// TwinCAT 3 PLC project plc_vat_test
// ProgramVersion: 3.1.4024.12
// libraries:
//   LCLS General, * (SLAC)
//   PMPS, * (SLAC - LCLS)
//   Tc2_EtherCAT, * (Beckhoff Automation GmbH)
//   Tc2_Math, * (Beckhoff Automation GmbH)
//   Tc2_Standard, * (Beckhoff Automation GmbH)
//   Tc2_System, * (Beckhoff Automation GmbH)
//   Tc2_Utilities, * (Beckhoff Automation GmbH)
//   Tc3_Module, * (Beckhoff Automation GmbH)
//   LCLS Vacuum,newest,SLAC - LCLS
// project tree:
//   DUTs/ ST_CoeParamsTest.TcDUT
//   DUTs/VAT590/EtherCAT Interface/ E_ControlMode.TcDUT, E_ControlModeSP.TcDUT (not stored), E_FatalErrors.TcDUT, ST_ExtendedWarnings.TcDUT (not stored), ST_GeneralControlSP.TcDUT (not stored), ST_GeneralStatus.TcDUT (not stored), ST_GeneralWarnings.TcDUT (not stored)
//   DUTs/VAT590/ E_VAT590_PID_CTRL.TcDUT (not stored), E_VAT590_PressureSensor.TcDUT (not stored), E_VCN_VAT590.TcDUT (not stored), E_VAT590_AccessMode.TcDUT (not stored), ST_CoEIndSub.TcDUT (not stored), ST_VAT590_COE.TcDUT, ST_VCN_VAT590.TcDUT, ST_VAT590_STATUS.TcDUT (not stored)
//   GVLs/ GVL_IO.TcGVL
//   / PlcTask.TcTTO
//   POUs/CoE/ FB_CoE_Read.TcPOU, FB_CoE_Write.TcPOU
//   POUs/Gauges/ FB_IE514.TcPOU, FB_MX7M.TcPOU
//   POUs/Valves/ FB_VCN_VAT590.TcPOU
//   POUs/ MAIN.TcPOU
// real-time tasks:
//   TASK PlcTask: cycle T#10ms, priority 20, ADS port 350
// I/O:
//   DEVICE Device 1 (EtherCAT), AmsNetId 172.21.132.149.2.1
//     Term 1 (EK1200) [EK1200-5000 EtherCAT Power supply (2A E-Bus)]
//       Term 3 (EL1004) [EL1004 4Ch. Dig. Input 24V, 3ms]
//       Term 5 (EL3174-0002) [EL3174-0002 4Ch. Ana. Input +/-10V, +/-20mA 16 Bit, Isolated Channels]
//       Term 10 (EL2624) [EL2624 4Ch. Relay Output, NO (125V AC / 30V DC)]
//       Term 8 (EK1110) [EK1110 EtherCAT extension]
//     VAT590_TEST [590 - All-metal variable leak valve]
// variable links:
//   plc_vat_test/plc_vat_test Instance <-> Device 1 (EtherCAT)/Term 1 (EK1200)/Term 10 (EL2624)
//     PlcTask Outputs/MAIN.fbIE514.q_xHV_DIS_CH1 <-> Channel 1/Output
//     PlcTask Outputs/MAIN.fbIE514.q_xHV_DIS_CH2 <-> Channel 2/Output
//     PlcTask Outputs/MAIN.fbMX7M.q_xHV_DIS <-> Channel 3/Output
//   plc_vat_test/plc_vat_test Instance <-> Device 1 (EtherCAT)/Term 1 (EK1200)/Term 3 (EL1004)
//     PlcTask Inputs/MAIN.fbIE514.i_xCH2_SEL <-> Channel 2/Input
//     PlcTask Inputs/MAIN.fbIE514.i_xERR_CH1 <-> Channel 3/Input
//     PlcTask Inputs/MAIN.fbIE514.i_xERR_CH2 <-> Channel 4/Input
//     PlcTask Inputs/MAIN.fbIE514.i_xHV_ON <-> Channel 1/Input
//   plc_vat_test/plc_vat_test Instance <-> Device 1 (EtherCAT)/Term 1 (EK1200)/Term 5 (EL3174-0002)
//     PlcTask Inputs/MAIN.fbIE514.i_iPRESS_R <-> AI Standard Channel 1/Value
//     PlcTask Inputs/MAIN.fbMX7M.i_iPRESS_R <-> AI Standard Channel 3/Value
//   plc_vat_test/plc_vat_test Instance <-> Device 1 (EtherCAT)/VAT590_TEST
//     PlcTask Inputs/MAIN.fbVCN590.i_bValveEthCatStatus <-> WcState/WcState
//     PlcTask Inputs/MAIN.fbVCN590.i_eControlMode <-> DI TxPDO-Map/Control mode
//     PlcTask Inputs/MAIN.fbVCN590.i_eFatalError <-> DI TxPDO-Map/Fatal error
//     PlcTask Inputs/MAIN.fbVCN590.i_nRawPosition <-> DI TxPDO-Map/Position
//     PlcTask Inputs/MAIN.fbVCN590.i_nRawPressure <-> DI TxPDO-Map/Pressure
//     PlcTask Inputs/MAIN.fbVCN590.i_stExtnWarnings <-> DI TxPDO-Map/Extended warnings
//     PlcTask Inputs/MAIN.fbVCN590.i_stGenStatus <-> DI TxPDO-Map/General status
//     PlcTask Inputs/MAIN.fbVCN590.i_stGenWarnings <-> DI TxPDO-Map/General warnings
//     PlcTask Inputs/MAIN.fbVCN590.i_stVat590PlcDriveRef/aNetId <-> InfoData/AdsAddr/netId
//     PlcTask Inputs/MAIN.fbVCN590.i_stVat590PlcDriveRef/nSlaveAddr <-> InfoData/AdsAddr/port
//     PlcTask Outputs/MAIN.fbVCN590.o_eCtrlModeSP <-> DO RxPDO-Map/Control mode setpoint
//     PlcTask Outputs/MAIN.fbVCN590.o_nRawPositionSP <-> DO RxPDO-Map/Position setpoint
//     PlcTask Outputs/MAIN.fbVCN590.o_nRawPressureSP <-> DO RxPDO-Map/Pressure setpoint
//     PlcTask Outputs/MAIN.fbVCN590.o_stGenCtrlSP <-> DO RxPDO-Map/General control setpoint

CONFIGURATION plc_vat_test
    RESOURCE PLC ON TwinCAT3
        TASK PlcTask(INTERVAL := T#10ms, PRIORITY := 20);
        PROGRAM MAIN WITH PlcTask : MAIN;
    END_RESOURCE
END_CONFIGURATION

// ---- DUTs/ST_CoeParamsTest.TcDUT
TYPE ST_CoeParamsTest :
STRUCT
	nWarnTemp : BYTE;
	nSwOffTemp : BYTE;
	nOffestA : INT;
	nOffestB : INT;
END_STRUCT
END_TYPE

// ---- DUTs/VAT590/EtherCAT Interface/E_ControlMode.TcDUT
{attribute 'qualified_only'}
{attribute 'strict'}
TYPE E_ControlMode :
(
	Init := 0,
	Synch := 1,
	ManualControl := 2,
	CloseValve := 3,
	OpenValve := 4,
	PressureControl := 5,
	HoldValve := 6,
	LearnProcedure := 7,
	InterlockOpen := 8,
	InterlockClose := 9,
	MaintenanceOpen := 10,
	MaintenanceClose := 11,
	PowerFailure := 12,
	Safety := 13,
	FatalError := 14
) USINT;
END_TYPE

// ---- DUTs/VAT590/EtherCAT Interface/E_FatalErrors.TcDUT
{attribute 'qualified_only'}
{attribute 'strict'}
TYPE E_FatalErrors :
(
	NO_FATAL_ERROR := 0,
	NoStopDetectedSynch := 20,
	ValveBlockedSynch := 21,
	ValveBlocked := 22,
	StepLossSynch := 25,
	MotorDriverFault := 40
) UINT;
END_TYPE

// ---- DUTs/VAT590/ST_VAT590_COE.TcDUT
TYPE ST_VAT590_COE :
STRUCT
	{attribute 'pytmc' := '
	pv: PID_CTRL
	io: io
	'}
	ePIDCtrl: E_VAT590_PID_CTRL;
	(*Adaptive Downstream Parameters*)
	{attribute 'pytmc' := '
    pv: SENS_DELAY_AD
	io: io
	field: EGU "s"
	field: DRVL 0.0
	field: DRVH 1.0
    '}
	fSensorDelay_AD : REAL;
	{attribute 'pytmc' := '
    pv: RAMP_TIME_AD
	io: io
	field: EGU "s"
	field: DRVL 0.0
	field: DRVH 1000000.0
    '}
	fRampTime_AD : REAL;
	{attribute 'pytmc' := '
    pv: RAMP_MODE_AD
	io: io
	field: ZNAM CONST_TIME
	field: ONAM CONST_SLOPE
    '}
	nRampMode_AD : BOOL;
	{attribute 'pytmc' := '
    pv: GAIN_FACTOR_AD
	io: io
	field: PREC 4
	field: DRVL 0.0001
	field: DRVH 7.5
    '}
	fGainFactor_AD : REAL;
	(*Fixed 1 Parameters*)
	{attribute 'pytmc' := '
    pv: RAMP_TIME_FIX1
	io: io
	field: EGU "s"
	field: DRVL 0.0
	field: DRVH 1000000.0
    '}
	fRampTime_FIX1 : REAL;
	{attribute 'pytmc' := '
    pv: RAMP_MODE_FIX1
	io: io
	field: ZNAM CONST_TIME
	field: ONAM CONST_SLOPE
    '}
	nRampMode_FIX1 : BOOL;
	{attribute 'pytmc' := '
    pv: CTRL_DIR_FIX1
	io: io
	field: ZNAM DOWNSTREAM
	field: ONAM UPSTREAM
    '}
	nCtrlDir_FIX1 : BOOL;
	{attribute 'pytmc' := '
    pv: PGAIN_FIX1
	io: io
	field: DRVL 0.001
	field: DRVH 100.0
    '}
	fPGain_FIX1 : REAL;
	{attribute 'pytmc' := '
    pv: IGAIN_FIX1
	io: io
	field: DRVL 0.0
	field: DRVH 100.0
    '}
	fIGain_FIX1 : REAL;
	(*Fixed 2 Parameters*)
	{attribute 'pytmc' := '
    pv: RAMP_TIME_FIX2
	io: io
	field: EGU "s"
	field: DRVL 0.0
	field: DRVH 1000000.0
    '}
	fRampTime_FIX2 : REAL;
	{attribute 'pytmc' := '
    pv: RAMP_MODE_FIX2
	io: io
	field: ZNAM CONST_TIME
	field: ONAM CONST_SLOPE
    '}
	nRampMode_FIX2 : BOOL;
	{attribute 'pytmc' := '
    pv: CTRL_DIR_FIX2
	io: io
	field: ZNAM DOWNSTREAM
	field: ONAM UPSTREAM
    '}
	nCtrlDir_FIX2 : BOOL;
	{attribute 'pytmc' := '
    pv: PGAIN_FIX2
	io: io
	field: DRVL 0.001
	field: DRVH 100.0
    '}
	fPGain_FIX2 : REAL;
	{attribute 'pytmc' := '
    pv: IGAIN_FIX2
	io: io
	field: DRVL 0.0
	field: DRVH 100.0
    '}
	fIGain_FIX2 : REAL;
	(*Soft Pump Parameters*)
	{attribute 'pytmc' := '
    pv: RAMP_TIME_SP
	io: io
	field: EGU "s"
	field: DRVL 0.0
	field: DRVH 1000000.0
    '}
	fRampTime_SP : REAL;
	{attribute 'pytmc' := '
    pv: RAMP_MODE_SP
	io: io
	field: ZNAM CONST_TIME
	field: ONAM CONST_SLOPE
    '}
	nRampMode_SP : BOOL;
	{attribute 'pytmc' := '
    pv: PGAIN_SP
	io: io
	field: DRVL 0.001
	field: DRVH 100.0
    '}
	fPGain_SP : REAL;
END_STRUCT
END_TYPE

// ---- DUTs/VAT590/ST_VCN_VAT590.TcDUT
TYPE ST_VCN_VAT590 :
STRUCT
	(* VCN - Valve Controlled Needle
	Used for VAT590 needle valves *)
	{attribute 'pytmc' := '
    pv: POS_RAW
	io: i
    '}
	nRawPosition : DINT; //Position readback
	{attribute 'pytmc' := '
    pv: PRES_RAW
	io: i
    '}
	nRawPressure : DINT; //Pressure readback
	{attribute 'pytmc' := '
    pv: PRES_TORR
	field: EGU "TORR"
	io: i
    '}
	fPressure : REAL; //Pressure readback in Torr units
	{attribute 'pytmc' := '
	pv: POS_SP
	io: i
	'}
	nPositionSP : DINT; //Position setpoint readback
	{attribute 'pytmc' := '
	pv: PRES_SP
	io: i
	'}
	nPressureSP : DINT; //Pressure setpoint readback
	{attribute 'pytmc' := '
    pv: ILK_OK
	field: ZNAM NOT OK
	field: ONAM OK
	field: ZSV MAJOR
	field: OSV NO_ALARM
	io: i
    '}
	bIlkOK : BOOL := FALSE; // Interlock Bit status
	{attribute 'pytmc' := '
    pv: POS_LIMIT
	io: io
	autosave_pass1: VAL DESC
    '}
	fPosSetLimit	: REAL := 100; // Percentage Upper limit on valve open
	{attribute 'pytmc' := '
    pv: PRES_SET_LIMIT
	io: io
	autosave_pass1: VAL DESC
    '}
	fPresSetLimit	: REAL := 1E-2; // Upper limit for pressure control 	
	{attribute 'pytmc' := '
    pv: PRES_RDBK_LIMIT
	io: io
	autosave_pass1: VAL DESC
    '}	
	fPresRdbkLimit : REAL := 1E-4;  //upper limit for pressure reading before valve close
	{attribute 'pytmc' := '
	pv: POS_REQ
	field: DRVL 0.0
	field: DRVH 100.0
	io: io
	'}
	fReqPosition : REAL; //Requested position (0.0-100.0%)
	{attribute 'pytmc' := '
	pv: PRES_REQ
	field: EGU "TORR"
	io: io;
	'}
	fReqPressure : REAL; //Requested pressure in Torr units
	{attribute 'pytmc' :=  ' 
	pv: STATE
	io: io
	'}
	eValveControl : E_VCN_VAT590; //Valve control mode
	{attribute 'pytmc' := '
    pv: 
	'}
	stValveStatus : ST_VAT590_STATUS; //All Valve status readbacks
	{attribute 'pytmc' :=  ' 
	pv: PRES_SENS
	io: io
	'}
	ePressureSensor : E_VAT590_PressureSensor; // Select pressure sensor
	{attribute 'pytmc' :=  ' 
	pv: REM_CTRL
	io: o
	'}
	eRemoteControl : E_VAT590_AccessMode; // Select remote control mode
	{attribute 'pytmc' := '
	pv: ZERO
	field: ZNAM NOT_ACTIVE
	field: ONAM ACTIVE
	io: o
	'}
	bZero : BOOL; // Activate Zero function bit
	{attribute 'pytmc' := '
    pv: 
	'}
	stCoeParameters : ST_VAT590_COE; //Coe Parameters
	{attribute 'pytmc' := '
	pv: COE_ERROR
	io: i
	field: ZNAM OK
	field: ONAM ERROR
	field: ZSV NO_ALARM
	field: OSV MAJOR
	'}
	bCoeError : BOOL; //Coe Interface Error
	{attribute 'pytmc' := '
	pv: COE_RESET
	io: io
	'}
	bResetCoeError : BOOL; //Reset Coe Interface
END_STRUCT
END_TYPE

// ---- GVLs/GVL_IO.TcGVL
{attribute 'qualified_only'}
VAR_GLOBAL
	//stPlcDriveRef AT %I*: ST_PlcDriveRef;
END_VAR

// ---- POUs/MAIN.TcPOU
PROGRAM MAIN
VAR
	
    {attribute 'pytmc' := '
      pv: VCN:TEST:01
    '}
	fbVCN590 : FB_VCN_VAT590; // Variable leak valve VAT590 function block
	fbMKS500 : FB_MKS500;
	
	stVG : ST_VG;
    {attribute 'pytmc' := '
      pv: GHC:TEST
    '}
	fbIE514 : FB_IE514;
	
    {attribute 'pytmc' := '
      pv: GCC:TEST
    '}
	fbMX7M : FB_MX7M;
	rPiraniPressure : REAL := 1E-4;
	
	rRealNumber : REAL := 8.367;
	intPart: INT;
    fracPart: REAL;
	rPressure : REAL := 0;
END_VAR

stVG.xPRESS_OK := TRUE;
stVG.rPress := rPiraniPressure;
fbMKS500.M_SetBits(30518);
fbMKS500(PG := stVG);

fbVCN590(bExtIlkOK := TRUE, IG := stVG);

fbIE514(PG := stVG);

fbMX7M(PG := stVG);

intPart := TRUNC_INT(rRealNumber); // Get the integer part
fracPart := LREAL_TO_REAL(FRAC(rRealNumber)); // Get the fractional part

rPressure := fracPart * LREAL_TO_REAL(EXPT(10,(intPart-11)));

END_PROGRAM

// ---- POUs/Valves/FB_VCN_VAT590.TcPOU
(* This function implements the Basic functions for the VAT590 needle valve*)
FUNCTION_BLOCK FB_VCN_VAT590 EXTENDS FB_Valve
VAR_INPUT
	bExtIlkOK : BOOL;        // External Interlock, SET to TRUE if not used
	IG : ST_VG;              // Input from a cold cathode gauge used in control loop
END_VAR
VAR_OUTPUT
	{attribute 'pytmc' := '
    pv:
	'}
	stVcnVat590	: ST_VCN_VAT590;       // Needle valve VAT590 structure
END_VAR
VAR CONSTANT
	cOpenPosition : REAL := 1E+5;      // Default position setpoint upper scale value
	cClosePosition : REAL := 0.0;      // Default position setpoint lower scale value
	cPresSPUpLim : REAL := 1E+6;       // Default pressure setpoint upper scale value
	cPresSPLowLim : REAL := 0;         // Default pressure setpoint lower scale value
	cPressCtrl : ST_CoEIndSub := (nIndex := 16#2199, nSubIndex := 0); // Selected pressure controller CoE register
	cSensorDelay_AD : ST_CoEIndSub := (nIndex := 16#219A, nSubIndex := 0); // Adaptive DS controller Sensor Delay CoE register
	cRampTime_AD : ST_CoEIndSub := (nIndex := 16#219B, nSubIndex := 0); // Adaptive DS controller Ramp Time CoE register
	cRampMode_AD : ST_CoEIndSub := (nIndex := 16#219C, nSubIndex := 0); // Adaptive DS controller Ramp Mode CoE register
	cGainFactor_AD : ST_CoEIndSub := (nIndex := 16#219E, nSubIndex := 0); // Adaptive DS controller Gain factor CoE register
	cRampTime_FIX1 : ST_CoEIndSub := (nIndex := 16#21A5, nSubIndex := 0); // Fixed 1 controller Ramp Time CoE register
	cRampMode_FIX1 : ST_CoEIndSub := (nIndex := 16#21A6, nSubIndex := 0); // Fixed 1 controller Ramp Mode CoE register
	cCtrlDir_FIX1 : ST_CoEIndSub := (nIndex := 16#21A7, nSubIndex := 0); // Fixed 1 controller Control Direction CoE register
	cPGain_FIX1 : ST_CoEIndSub := (nIndex := 16#21A8, nSubIndex := 0); // Fixed 1 controller P Gain CoE register
	cIGain_FIX1 : ST_CoEIndSub := (nIndex := 16#21A9, nSubIndex := 0); // Fixed 1 controller I Gain CoE register
	cRampTime_FIX2 : ST_CoEIndSub := (nIndex := 16#21AF, nSubIndex := 0); // Fixed 2 controller Ramp Time CoE register
	cRampMode_FIX2 : ST_CoEIndSub := (nIndex := 16#21B0, nSubIndex := 0); // Fixed 2 controller Ramp Mode CoE register
	cCtrlDir_FIX2 : ST_CoEIndSub := (nIndex := 16#21B1, nSubIndex := 0); // Fixed 2 controller Control Direction CoE register
	cPGain_FIX2 : ST_CoEIndSub := (nIndex := 16#21B2, nSubIndex := 0); // Fixed 2 controller P Gain CoE register
	cIGain_FIX2 : ST_CoEIndSub := (nIndex := 16#21B3, nSubIndex := 0); // Fixed 2 controller I Gain CoE register
	cRampTime_SP : ST_CoEIndSub := (nIndex := 16#21B9, nSubIndex := 0); // Soft Pump controller Ramp Time CoE register
	cRampMode_SP : ST_CoEIndSub := (nIndex := 16#21BA, nSubIndex := 0); // Soft Pump controller Ramp Time CoE register
	cPGain_SP : ST_CoEIndSub := (nIndex := 16#21BC, nSubIndex := 0); // Soft Pump controller Ramp Time CoE register
END_VAR
VAR
	fCalcPosSP : REAL := 0;
	fCalcPresSP : REAL := 0;
	eValveModeSP : E_ControlModeSP;
	fReqPos : REAL;                    // Requested position internal variable
	fReqPres : REAL;                   // Requested pressure internal variable
	fPresLowLim : REAL := 1E-10;       // Pressure sensor lower scale value
	fSlope : REAL := 1E+5;             // Slope (Units per decade) used for conversion from Torr units
	fVbase : REAL := 1E+5;             // Vbase (Units per decade) defined for how much the curve is shifted
	bRemAcsToggle : BOOL;              // Remote access control bit
	//timer for zero function 
	tZeroTogg : TON := (PT := T#1S);
	//timer for remote function
	tRemAcsTogg : TON := (PT := T#500MS);
	//used for logging
	ePreviousState : E_VCN_VAT590;
	
	(*CoE Interface*)
	(*Link this to your VAT590 reference variables under InfoData.*)
	stVat590PlcDriveRef AT %I*: ST_PlcDriveRef;
	stVat590DriveRef : ST_DriveRef := (
		sNetId := F_CreateAmsNetId(stVat590PlcDriveRef.aNetId),
		nSlaveAddr := stVat590PlcDriveRef.nSlaveAddr,
		nDriveNo := stVat590PlcDriveRef.nDriveNo,
		nDriveType := stVat590PlcDriveRef.nDriveType
	);

	fbCoeRead : FB_CoERead_ByDriveRef := (
		stDriveRef := stVat590DriveRef
	);
	fbCoeWrite : FB_CoEWrite_ByDriveRef := (
		stDriveRef := stVat590DriveRef
	);
	
	stCoeParameters : ST_VAT590_COE;   //Internal storage of CoE parameters
	nCaseReadCoe : UINT := 1;          //Iterator for going through all CoE parameters
	rtCoeReset : R_TRIG;               //Rising edge trigger for reset CoE Interface error
	ftCoeReadBusy : F_TRIG;            //Falling edge trigger for CoE read new data
	ftCoeWriteBusy : F_TRIG;           //Falling edge trigger for CoE write data
	bFirstRead : BOOL := TRUE;
	
	(*VAT590 Ethercat IO Interface*)
	//Ethercat Interface Inputs
	i_nRawPosition       AT %I* : DINT;               // Position readback from the valve
	i_nRawPressure       AT %I* : DINT;               // Pressure readback from the valve
	i_eControlMode       AT %I* : E_ControlMode;      // Valve control mode readback
	i_eFatalError        AT %I* : E_FatalErrors;      // Valve Fatal Errors readback
	i_stGenStatus        AT %I* : ST_GeneralStatus;   // Valve General Status readback
	i_stGenWarnings      AT %I* : ST_GeneralWarnings; // Valve General Warnings readback
	i_stExtnWarnings     AT %I* : ST_ExtendedWarnings;// Valve Extended Warnings readback
	//Ethercat Interface Outputs
	o_nRawPositionSP     AT %Q* : DINT;               // Position setpoint
	o_nRawPressureSP     AT %Q* : DINT;               // Pressure setpoint
	o_eCtrlModeSP        AT %Q* : E_ControlModeSP;    // Valve control mode setpoint
	o_stGenCtrlSP        AT %Q* : ST_GeneralControlSP;// General Control setpoint
END_VAR
VAR PERSISTENT
    fUpperLimit	: REAL;                // Max position in % that can be requested
	fPresMaxLim : REAL;                // Max pressure in Torr that can be requested
	fPresRbMaxLim : REAL;               // Max pressure in Torr read by chamber gauge, valve will close above the pressure.
END_VAR

(* Needle valve control FB
J. Govednik 2021-11-22

This FB should be used as a low level control block.

It provides:
Valve position ceiling
Interlock
Scaling

It could be used for:
Valve position/flow linearization
*)

(*Read from EPICS and Valve Ethercat interface*)
ReadFromInput();

(*Checking which Control mode is selected*)
IF bExtIlkOK THEN
	CASE stVcnVat590.eValveControl OF
		E_VCN_VAT590.OpenValve:
			eValveModeSP := E_ControlModeSP.OpenValve;
		E_VCN_VAT590.CloseValve:
			eValveModeSP := E_ControlModeSP.CloseValve;
		E_VCN_VAT590.ManualControl:
		    IF IG.xPRESS_OK AND IG.rPRESS <= fPresRbMaxLim THEN
				eValveModeSP := E_ControlModeSP.ManualControl;
			ELSE
				eValveModeSP := E_ControlModeSP.CloseValve; // Close valve if something is wrong with the gauge
				stVcnVat590.eValveControl := E_VCN_VAT590.CloseValve;
			END_IF	
		E_VCN_VAT590.PressureControl:
			IF IG.xPRESS_OK AND IG.rPRESS <= fPresRbMaxLim THEN
				eValveModeSP := E_ControlModeSP.PressureControl;
			ELSE
				eValveModeSP := E_ControlModeSP.CloseValve; // Close valve if something is wrong with the gauge
				stVcnVat590.eValveControl := E_VCN_VAT590.CloseValve;
			END_IF
		E_VCN_VAT590.HoldValve:
			IF stVcnVat590.stValveStatus.eControlMode = E_ControlMode.ManualControl OR
				stVcnVat590.stValveStatus.eControlMode = E_ControlMode.PressureControl THEN
				eValveModeSP := E_ControlModeSP.HoldValve;
			END_IF
	END_CASE
ELSE
	fReqPos := 0;
	eValveModeSP := E_ControlModeSP.CloseValve;
	stVcnVat590.eValveControl := E_VCN_VAT590.CloseValve;
END_IF

(*Requested Position calculation*)
fReqPos := LIMIT(0, fReqPos, fUpperLimit);
fCalcPosSP := fReqPos * (cOpenPosition-cClosePosition)/100 + cClosePosition;
fCalcPosSP := LIMIT(cClosePosition, fCalcPosSP, cOpenPosition); //The requested position SP should remain within this range

(*Pressure calculation*)
//Limit the input from EPICS between upper and lower limit defined for seleceted pressure sensor
fReqPres := LIMIT(fPresLowLim, fReqPres, fPresMaxLim);

// Calculate pressure readback and pressure setpoint according to selected pressure gauge
CASE stVcnVat590.ePressureSensor OF
	E_VAT590_PressureSensor.MKS500:
		fPresLowLim := 1.0E-10;
		fSlope := 1E+5;
		fVbase := 1E+5;
		//Calcuate pressure setpoint
		fCalcPresSP := fSlope * LOG(fReqPres/fPresLowLim) + fVbase;
		fCalcPresSP := LIMIT(cPresSPLowLim, fCalcPresSP, cPresSPUpLim); //The requested pressure SP should remain within this range
		//Calculate pressure readback in Torr units
		stVcnVat590.fPressure := LREAL_TO_REAL(EXPT(10,((DINT_TO_REAL(i_nRawPressure)-fVbase)/fSlope + LOG(fPresLowLim))));
	ELSE
		fCalcPresSP := 0;
		stVcnVat590.fPressure := 0;
END_CASE

(*Calculated Pressure SP and Pressure readback is 0 if Pressure sensor is not working*) 
IF NOT (IG.xPRESS_OK AND IG.rPRESS < fPresRbMaxLim ) THEN
	fCalcPresSP := 0;
	stVcnVat590.fPressure := 0;
END_IF

(*Zero function*)
IF stVcnVat590.stValveStatus.bZeroDisabled OR tZeroTogg.Q THEN
	stVcnVat590.bZero := FALSE;
END_IF
tZeroTogg.IN := stVcnVat590.bZero;
tZeroTogg();

(*Set Remote Access*)
IF stVcnVat590.stValveStatus.eRemoteStatus <> stVcnVat590.eRemoteControl THEN
	tRemAcsTogg.IN := TRUE;
	IF tRemAcsTogg.Q THEN
		bRemAcsToggle := NOT bRemAcsToggle;
		tRemAcsTogg.IN := FALSE;
	END_IF
END_IF
tRemAcsTogg();

(*Reset Coe Interface error*)
rtCoeReset(CLK := stVcnVat590.bResetCoeError);
IF rtCoeReset.Q THEN
	stVcnVat590.bResetCoeError := FALSE;
END_IF

(*Read CoE Parameters*)
ReadCoeParameters();

(*Write CoE Parameters*)
WriteCoeParameters();

(*Write to EPICS and Valve Ethercat interface*)
WriteToOutput();

(*Load or save the persistent variables*)
LoadPersistentData();

(*Logging*)
Logger();

ACTION LoadPersistentData:
(*On first PLC pass, load the persistent value into the structrue variable*)
IF (bRestorePersistentData) THEN
	bRestorePersistentData	:= FALSE;
	IF (fUpperLimit <> 0) THEN
		stVcnVat590.fPosSetLimit := fUpperLimit;
	END_IF;
	IF (fPresMaxLim <> 0) THEN
		stVcnVat590.fPresSetLimit := fPresMaxLim;
	END_IF;
	IF (fPresRbMaxLim <> 0) THEN
		stVcnVat590.fPresRdbkLimit := fPresRbMaxLim;
	END_IF;    
END_IF
END_ACTION

ACTION Logger:
// ILK logger
IF NOT (stVcnVat590.bIlkOK ) AND NOT(ePreviousState = E_VCN_VAT590.CloseValve) THEN
 		fbLogger(sMsg:='Lost interlock ok bit while valve was open.', eSevr:=TcEventSeverity.Critical);  	
END_IF


//Control STATE Logger  
IF ePreviousState <> stVcnVat590.eValveControl THEN
	  CASE stVcnVat590.eValveControl OF
		E_VCN_VAT590.ManualControl:
			fbLogger(sMsg:='Valve in manual control mode.', eSevr:=TcEventSeverity.Warning);
		E_VCN_VAT590.HoldValve:
			fbLogger(sMsg:='Valve in hold control mode.', eSevr:=TcEventSeverity.Warning);
		E_VCN_VAT590.OpenValve:
			fbLogger(sMsg:='Valve Open.', eSevr:=TcEventSeverity.Info);
		E_VCN_VAT590.PressureControl:
			fbLogger(sMsg:='Valve in pressure control mode.', eSevr:=TcEventSeverity.Info);
		E_VCN_VAT590.CloseValve:
			fbLogger(sMsg:='Valve closed.', eSevr:=TcEventSeverity.Info);
	  END_CASE
	  ePreviousState := stVcnVat590.eValveControl;  
  END_IF
 

// Log valve open
tAction(CLK:= (stVcnVat590.eValveControl = E_VCN_VAT590.OpenValve) );
IF tAction.Q THEN fbLogger(sMsg:='Valve commanded to fully open', eSevr:=TcEventSeverity.Info); END_IF
END_ACTION

ACTION ReadCoeParameters:
CASE nCaseReadCoe OF
	0:
		//fbCoeRead.bExecute := FALSE;
		stVcnVat590.bCoeError := TRUE;
		IF rtCoeReset.Q THEN
			nCaseReadCoe := 1;
			stVcnVat590.bCoeError := FALSE;
			bFirstRead := TRUE; // Set bFirstRead after Coe interface reset
		END_IF
	1:
		fbCoeRead.nIndex := cPressCtrl.nIndex;
		fbCoeRead.nSubIndex := cPressCtrl.nSubIndex;
		fbCoeRead.pDstBuf := ADR(stVcnVat590.stCoeInterface.nPressCtrl);
		fbCoeRead.cbBufLen := SIZEOF(stVcnVat590.stCoeInterface.nPressCtrl);
		fbCoeRead.bExecute := TRUE;
	2:
		fbCoeRead.nIndex := cSensorDelay_AD.nIndex;
		fbCoeRead.nSubIndex := cSensorDelay_AD.nSubIndex;
		fbCoeRead.pDstBuf := ADR(stVcnVat590.stCoeInterface.fSensorDelay_AD);
		fbCoeRead.cbBufLen := SIZEOF(stVcnVat590.stCoeInterface.fSensorDelay_AD);
		fbCoeRead.bExecute := TRUE;
	3:
		fbCoeRead.nIndex := cRampTime_AD.nIndex;
		fbCoeRead.nSubIndex := cRampTime_AD.nSubIndex;
		fbCoeRead.pDstBuf := ADR(stVcnVat590.stCoeInterface.fRampTime_AD);
		fbCoeRead.cbBufLen := SIZEOF(stVcnVat590.stCoeInterface.fRampTime_AD);
		fbCoeRead.bExecute := TRUE;
	4:
		fbCoeRead.nIndex := cRampMode_AD.nIndex;
		fbCoeRead.nSubIndex := cRampMode_AD.nSubIndex;
		fbCoeRead.pDstBuf := ADR(stVcnVat590.stCoeInterface.nRampMode_AD);
		fbCoeRead.cbBufLen := SIZEOF(stVcnVat590.stCoeInterface.nRampMode_AD);
		fbCoeRead.bExecute := TRUE;
	5:
		fbCoeRead.nIndex := cGainFactor_AD.nIndex;
		fbCoeRead.nSubIndex := cGainFactor_AD.nSubIndex;
		fbCoeRead.pDstBuf := ADR(stVcnVat590.stCoeInterface.fGainFactor_AD);
		fbCoeRead.cbBufLen := SIZEOF(stVcnVat590.stCoeInterface.fGainFactor_AD);
		fbCoeRead.bExecute := TRUE;
	6:
		fbCoeRead.nIndex := cRampTime_FIX1.nIndex;
		fbCoeRead.nSubIndex := cRampTime_FIX1.nSubIndex;
		fbCoeRead.pDstBuf := ADR(stVcnVat590.stCoeInterface.fRampTime_FIX1);
		fbCoeRead.cbBufLen := SIZEOF(stVcnVat590.stCoeInterface.fRampTime_FIX1);
		fbCoeRead.bExecute := TRUE;
	7:
		fbCoeRead.nIndex := cRampMode_FIX1.nIndex;
		fbCoeRead.nSubIndex := cRampMode_FIX1.nSubIndex;
		fbCoeRead.pDstBuf := ADR(stVcnVat590.stCoeInterface.nRampMode_FIX1);
		fbCoeRead.cbBufLen := SIZEOF(stVcnVat590.stCoeInterface.nRampMode_FIX1);
		fbCoeRead.bExecute := TRUE;
	8:
		fbCoeRead.nIndex := cCtrlDir_FIX1.nIndex;
		fbCoeRead.nSubIndex := cCtrlDir_FIX1.nSubIndex;
		fbCoeRead.pDstBuf := ADR(stVcnVat590.stCoeInterface.nCtrlDir_FIX1);
		fbCoeRead.cbBufLen := SIZEOF(stVcnVat590.stCoeInterface.nCtrlDir_FIX1);
		fbCoeRead.bExecute := TRUE;
	9:
		fbCoeRead.nIndex := cPGain_FIX1.nIndex;
		fbCoeRead.nSubIndex := cPGain_FIX1.nSubIndex;
		fbCoeRead.pDstBuf := ADR(stVcnVat590.stCoeInterface.fPGain_FIX1);
		fbCoeRead.cbBufLen := SIZEOF(stVcnVat590.stCoeInterface.fPGain_FIX1);
		fbCoeRead.bExecute := TRUE;
	10:
		fbCoeRead.nIndex := cIGain_FIX1.nIndex;
		fbCoeRead.nSubIndex := cIGain_FIX1.nSubIndex;
		fbCoeRead.pDstBuf := ADR(stVcnVat590.stCoeInterface.fIGain_FIX1);
		fbCoeRead.cbBufLen := SIZEOF(stVcnVat590.stCoeInterface.fIGain_FIX1);
		fbCoeRead.bExecute := TRUE;
	11:
		fbCoeRead.nIndex := cRampTime_FIX2.nIndex;
		fbCoeRead.nSubIndex := cRampTime_FIX2.nSubIndex;
		fbCoeRead.pDstBuf := ADR(stVcnVat590.stCoeInterface.fRampTime_FIX2);
		fbCoeRead.cbBufLen := SIZEOF(stVcnVat590.stCoeInterface.fRampTime_FIX2);
		fbCoeRead.bExecute := TRUE;
	12:
		fbCoeRead.nIndex := cRampMode_FIX2.nIndex;
		fbCoeRead.nSubIndex := cRampMode_FIX2.nSubIndex;
		fbCoeRead.pDstBuf := ADR(stVcnVat590.stCoeInterface.nRampMode_FIX2);
		fbCoeRead.cbBufLen := SIZEOF(stVcnVat590.stCoeInterface.nRampMode_FIX2);
		fbCoeRead.bExecute := TRUE;
	13:
		fbCoeRead.nIndex := cCtrlDir_FIX2.nIndex;
		fbCoeRead.nSubIndex := cCtrlDir_FIX2.nSubIndex;
		fbCoeRead.pDstBuf := ADR(stVcnVat590.stCoeInterface.nCtrlDir_FIX2);
		fbCoeRead.cbBufLen := SIZEOF(stVcnVat590.stCoeInterface.nCtrlDir_FIX2);
		fbCoeRead.bExecute := TRUE;
	14:
		fbCoeRead.nIndex := cPGain_FIX2.nIndex;
		fbCoeRead.nSubIndex := cPGain_FIX2.nSubIndex;
		fbCoeRead.pDstBuf := ADR(stVcnVat590.stCoeInterface.fPGain_FIX2);
		fbCoeRead.cbBufLen := SIZEOF(stVcnVat590.stCoeInterface.fPGain_FIX2);
		fbCoeRead.bExecute := TRUE;
	15:
		fbCoeRead.nIndex := cIGain_FIX2.nIndex;
		fbCoeRead.nSubIndex := cIGain_FIX2.nSubIndex;
		fbCoeRead.pDstBuf := ADR(stVcnVat590.stCoeInterface.fIGain_FIX2);
		fbCoeRead.cbBufLen := SIZEOF(stVcnVat590.stCoeInterface.fIGain_FIX2);
		fbCoeRead.bExecute := TRUE;
	16:
		fbCoeRead.nIndex := cRampTime_SP.nIndex;
		fbCoeRead.nSubIndex := cRampTime_SP.nSubIndex;
		fbCoeRead.pDstBuf := ADR(stVcnVat590.stCoeInterface.fRampTime_SP);
		fbCoeRead.cbBufLen := SIZEOF(stVcnVat590.stCoeInterface.fRampTime_SP);
		fbCoeRead.bExecute := TRUE;
	17:
		fbCoeRead.nIndex := cRampMode_SP.nIndex;
		fbCoeRead.nSubIndex := cRampMode_SP.nSubIndex;
		fbCoeRead.pDstBuf := ADR(stVcnVat590.stCoeInterface.nRampMode_SP);
		fbCoeRead.cbBufLen := SIZEOF(stVcnVat590.stCoeInterface.nRampMode_SP);
		fbCoeRead.bExecute := TRUE;
	18:
		fbCoeRead.nIndex := cPGain_SP.nIndex;
		fbCoeRead.nSubIndex := cPGain_SP.nSubIndex;
		fbCoeRead.pDstBuf := ADR(stVcnVat590.stCoeInterface.fPGain_SP);
		fbCoeRead.cbBufLen := SIZEOF(stVcnVat590.stCoeInterface.fPGain_SP);
		fbCoeRead.bExecute := TRUE;
END_CASE

ftCoeReadBusy(CLK:=fbCoeRead.bBusy);

IF ftCoeReadBusy.Q THEN
	fbCoeRead.bExecute := FALSE;
	IF NOT fbCoeRead.bError THEN
		nCaseReadCoe := nCaseReadCoe + 1;
		IF nCaseReadCoe > 18 THEN
			nCaseReadCoe := 1;
			bFirstRead := FALSE; // Reset bFirstRead after successfull readout of all parameters
		END_IF
	END_IF
END_IF

fbCoeRead();
stCoeParameters := stVcnVat590.stCoeInterface; //Save current values to internal structure
END_ACTION

ACTION ReadFromInput:
(*Read from EPICS*)
fUpperLimit := LIMIT(0, stVcnVat590.fPosSetLimit, 100);
fPresMaxLim := LIMIT(1.0E-10, stVcnVat590.fPresSetLimit, 1.0E-2);
fPresRbMaxLim := LIMIT(1.0E-10, stVcnVat590.fPresRdbkLimit, 1.0E-2);
fReqPos := LIMIT(0, stVcnVat590.fReqPosition, 100);
fReqPres := LIMIT(1.0E-10, stVcnVat590.fReqPressure, 1.0E-2);

(*Read from VAT valve*)
stVcnVat590.stValveStatus.eControlMode := i_eControlMode;
stVcnVat590.stValveStatus.eFatalErrors := i_eFatalError;
stVcnVat590.nRawPosition := i_nRawPosition;
stVcnVat590.nRawPressure := i_nRawPressure;
//Mapping General statuses
stVcnVat590.stValveStatus.bFieldBusDatavalid := i_stGenStatus.Bit0FieldBusDatavalid;
stVcnVat590.stValveStatus.bZeroExecuted := i_stGenStatus.Bit1ZeroExecuted;
stVcnVat590.stValveStatus.bPingPongRxBit := i_stGenStatus.Bit2PingPongRxBit;
stVcnVat590.stValveStatus.bPressureSimulation := i_stGenStatus.Bit3PressureSimulation;
stVcnVat590.stValveStatus.bPressureSPReached := i_stGenStatus.Bit4PressureSPReached;
stVcnVat590.stValveStatus.bWarningsActive := i_stGenStatus.Bit9WarningsActive;
//Read Remote status 
stVcnVat590.stValveStatus.eRemoteStatus.0 := i_stGenStatus.Bit7AccessModeBit0;
stVcnVat590.stValveStatus.eRemoteStatus.1 := i_stGenStatus.Bit8AccessModeBit1;
//Mapping General warnings
stVcnVat590.stValveStatus.bServiceRequest := i_stGenWarnings.Bit0ServiceRequest;
stVcnVat590.stValveStatus.bPowerFailureBattery := i_stGenWarnings.Bit3PowerFailureBattery;
stVcnVat590.stValveStatus.bSensMeasUnitFault := i_stGenWarnings.Bit10SensMeasUnitFault;
//Mapping Extended warnings
stVcnVat590.stValveStatus.bRemoteControlNotPossible := i_stExtnWarnings.Bit0RemoteControlNotPossible;
stVcnVat590.stValveStatus.bControlModeSPNotAllowed := i_stExtnWarnings.Bit1ControlModeSPNotAllowed;
stVcnVat590.stValveStatus.bZeroDisabled := i_stExtnWarnings.Bit2ZeroDisabled;
stVcnVat590.stValveStatus.bPFODeactivated := i_stExtnWarnings.Bit3PFODeactivated;
stVcnVat590.stValveStatus.bPressureSPOutOfRange := i_stExtnWarnings.Bit5PressureSPOutOfRange;
stVcnVat590.stValveStatus.bPositionSPOutOfRange := i_stExtnWarnings.Bit6PositionSPOutOfRange;
stVcnVat590.stValveStatus.bCtrlSPOutOfRange := i_stExtnWarnings.Bit10CtrlSPOutOfRange;
stVcnVat590.stValveStatus.bGeneralCtrlSPOutOfRange := i_stExtnWarnings.Bit11GeneralCtrlSPOutOfRange;
stVcnVat590.stValveStatus.bProcDataSettingsNotvalid := i_stExtnWarnings.Bit12ProcDataSettingsNotvalid;
END_ACTION

METHOD SetThrottle : BOOL
VAR_INPUT
	rUpperLimit	:	REAL;
END_VAR
stVcnVat590.fPosSetLimit := LIMIT(0, rUpperLimit, 100);
END_METHOD

METHOD ValveControl : BOOL
VAR_INPUT
	state : E_VCN_VAT590; // Set Control modes
END_VAR
stVcnVat590.eValveControl := state;
END_METHOD

ACTION WriteCoeParameters:
// User will change one parameter at a time so solution with ELSIF should work OK
IF stVcnVat590.bCoeError THEN
	//fbCoeWrite.bExecute := FALSE;
	IF rtCoeReset.Q THEN
		stVcnVat590.bCoeError := FALSE;
	END_IF;
ELSIF bFirstRead THEN
	;//Wait until first first readout of all CoE parameters is completed
ELSIF stVcnVat590.stCoeInterface.nPressCtrl <> stCoeParameters.nPressCtrl THEN
	fbCoeWrite.nIndex := cPressCtrl.nIndex;
	fbCoeWrite.nSubIndex := cPressCtrl.nSubIndex;
	fbCoeWrite.pSrcBuf := ADR(stVcnVat590.stCoeInterface.nPressCtrl);
	fbCoeWrite.cbBufLen := SIZEOF(stVcnVat590.stCoeInterface.nPressCtrl);
	fbCoeWrite.bExecute := TRUE;
ELSIF stVcnVat590.stCoeInterface.fSensorDelay_AD <> stCoeParameters.fSensorDelay_AD THEN
	fbCoeWrite.nIndex := cSensorDelay_AD.nIndex;
	fbCoeWrite.nSubIndex := cSensorDelay_AD.nSubIndex;
	fbCoeWrite.pSrcBuf := ADR(stVcnVat590.stCoeInterface.fSensorDelay_AD);
	fbCoeWrite.cbBufLen := SIZEOF(stVcnVat590.stCoeInterface.fSensorDelay_AD);
	fbCoeWrite.bExecute := TRUE;
ELSIF stVcnVat590.stCoeInterface.fRampTime_AD <> stCoeParameters.fRampTime_AD THEN
	fbCoeWrite.nIndex := cRampTime_AD.nIndex;
	fbCoeWrite.nSubIndex := cRampTime_AD.nSubIndex;
	fbCoeWrite.pSrcBuf := ADR(stVcnVat590.stCoeInterface.fRampTime_AD);
	fbCoeWrite.cbBufLen := SIZEOF(stVcnVat590.stCoeInterface.fRampTime_AD);
	fbCoeWrite.bExecute := TRUE;
ELSIF stVcnVat590.stCoeInterface.nRampMode_AD <> stCoeParameters.nRampMode_AD THEN
	fbCoeWrite.nIndex := cRampMode_AD.nIndex;
	fbCoeWrite.nSubIndex := cRampMode_AD.nSubIndex;
	fbCoeWrite.pSrcBuf := ADR(stVcnVat590.stCoeInterface.nRampMode_AD);
	fbCoeWrite.cbBufLen := SIZEOF(stVcnVat590.stCoeInterface.nRampMode_AD);
	fbCoeWrite.bExecute := TRUE;
ELSIF stVcnVat590.stCoeInterface.fGainFactor_AD <> stCoeParameters.fGainFactor_AD THEN
	fbCoeWrite.nIndex := cGainFactor_AD.nIndex;
	fbCoeWrite.nSubIndex := cGainFactor_AD.nSubIndex;
	fbCoeWrite.pSrcBuf := ADR(stVcnVat590.stCoeInterface.fGainFactor_AD);
	fbCoeWrite.cbBufLen := SIZEOF(stVcnVat590.stCoeInterface.fGainFactor_AD);
	fbCoeWrite.bExecute := TRUE;
ELSIF stVcnVat590.stCoeInterface.fRampTime_FIX1 <> stCoeParameters.fRampTime_FIX1 THEN
	fbCoeWrite.nIndex := cRampTime_FIX1.nIndex;
	fbCoeWrite.nSubIndex := cRampTime_FIX1.nSubIndex;
	fbCoeWrite.pSrcBuf := ADR(stVcnVat590.stCoeInterface.fRampTime_FIX1);
	fbCoeWrite.cbBufLen := SIZEOF(stVcnVat590.stCoeInterface.fRampTime_FIX1);
	fbCoeWrite.bExecute := TRUE;
ELSIF stVcnVat590.stCoeInterface.nRampMode_FIX1 <> stCoeParameters.nRampMode_FIX1 THEN
	fbCoeWrite.nIndex := cRampMode_FIX1.nIndex;
	fbCoeWrite.nSubIndex := cRampMode_FIX1.nSubIndex;
	fbCoeWrite.pSrcBuf := ADR(stVcnVat590.stCoeInterface.nRampMode_FIX1);
	fbCoeWrite.cbBufLen := SIZEOF(stVcnVat590.stCoeInterface.nRampMode_FIX1);
	fbCoeWrite.bExecute := TRUE;
ELSIF stVcnVat590.stCoeInterface.nCtrlDir_FIX1 <> stCoeParameters.nCtrlDir_FIX1 THEN
	fbCoeWrite.nIndex := cCtrlDir_FIX1.nIndex;
	fbCoeWrite.nSubIndex := cCtrlDir_FIX1.nSubIndex;
	fbCoeWrite.pSrcBuf := ADR(stVcnVat590.stCoeInterface.nCtrlDir_FIX1);
	fbCoeWrite.cbBufLen := SIZEOF(stVcnVat590.stCoeInterface.nCtrlDir_FIX1);
	fbCoeWrite.bExecute := TRUE;
ELSIF stVcnVat590.stCoeInterface.fPGain_FIX1 <> stCoeParameters.fPGain_FIX1 THEN
	fbCoeWrite.nIndex := cPGain_FIX1.nIndex;
	fbCoeWrite.nSubIndex := cPGain_FIX1.nSubIndex;
	fbCoeWrite.pSrcBuf := ADR(stVcnVat590.stCoeInterface.fPGain_FIX1);
	fbCoeWrite.cbBufLen := SIZEOF(stVcnVat590.stCoeInterface.fPGain_FIX1);
	fbCoeWrite.bExecute := TRUE;
ELSIF stVcnVat590.stCoeInterface.fIGain_FIX1 <> stCoeParameters.fIGain_FIX1 THEN
	fbCoeWrite.nIndex := cIGain_FIX1.nIndex;
	fbCoeWrite.nSubIndex := cIGain_FIX1.nSubIndex;
	fbCoeWrite.pSrcBuf := ADR(stVcnVat590.stCoeInterface.fIGain_FIX1);
	fbCoeWrite.cbBufLen := SIZEOF(stVcnVat590.stCoeInterface.fIGain_FIX1);
	fbCoeWrite.bExecute := TRUE;
ELSIF stVcnVat590.stCoeInterface.fRampTime_FIX2 <> stCoeParameters.fRampTime_FIX2 THEN
	fbCoeWrite.nIndex := cRampTime_FIX2.nIndex;
	fbCoeWrite.nSubIndex := cRampTime_FIX2.nSubIndex;
	fbCoeWrite.pSrcBuf := ADR(stVcnVat590.stCoeInterface.fRampTime_FIX2);
	fbCoeWrite.cbBufLen := SIZEOF(stVcnVat590.stCoeInterface.fRampTime_FIX2);
	fbCoeWrite.bExecute := TRUE;
ELSIF stVcnVat590.stCoeInterface.nRampMode_FIX2 <> stCoeParameters.nRampMode_FIX2 THEN
	fbCoeWrite.nIndex := cRampMode_FIX2.nIndex;
	fbCoeWrite.nSubIndex := cRampMode_FIX2.nSubIndex;
	fbCoeWrite.pSrcBuf := ADR(stVcnVat590.stCoeInterface.nRampMode_FIX2);
	fbCoeWrite.cbBufLen := SIZEOF(stVcnVat590.stCoeInterface.nRampMode_FIX2);
	fbCoeWrite.bExecute := TRUE;
ELSIF stVcnVat590.stCoeInterface.nCtrlDir_FIX2 <> stCoeParameters.nCtrlDir_FIX2 THEN
	fbCoeWrite.nIndex := cCtrlDir_FIX2.nIndex;
	fbCoeWrite.nSubIndex := cCtrlDir_FIX2.nSubIndex;
	fbCoeWrite.pSrcBuf := ADR(stVcnVat590.stCoeInterface.nCtrlDir_FIX2);
	fbCoeWrite.cbBufLen := SIZEOF(stVcnVat590.stCoeInterface.nCtrlDir_FIX2);
	fbCoeWrite.bExecute := TRUE;
ELSIF stVcnVat590.stCoeInterface.fPGain_FIX2 <> stCoeParameters.fPGain_FIX2 THEN
	fbCoeWrite.nIndex := cPGain_FIX2.nIndex;
	fbCoeWrite.nSubIndex := cPGain_FIX2.nSubIndex;
	fbCoeWrite.pSrcBuf := ADR(stVcnVat590.stCoeInterface.fPGain_FIX2);
	fbCoeWrite.cbBufLen := SIZEOF(stVcnVat590.stCoeInterface.fPGain_FIX2);
	fbCoeWrite.bExecute := TRUE;
ELSIF stVcnVat590.stCoeInterface.fIGain_FIX2 <> stCoeParameters.fIGain_FIX2 THEN
	fbCoeWrite.nIndex := cIGain_FIX2.nIndex;
	fbCoeWrite.nSubIndex := cIGain_FIX2.nSubIndex;
	fbCoeWrite.pSrcBuf := ADR(stVcnVat590.stCoeInterface.fIGain_FIX2);
	fbCoeWrite.cbBufLen := SIZEOF(stVcnVat590.stCoeInterface.fIGain_FIX2);
	fbCoeWrite.bExecute := TRUE;
ELSIF stVcnVat590.stCoeInterface.fRampTime_SP <> stCoeParameters.fRampTime_SP THEN
	fbCoeWrite.nIndex := cRampTime_SP.nIndex;
	fbCoeWrite.nSubIndex := cRampTime_SP.nSubIndex;
	fbCoeWrite.pSrcBuf := ADR(stVcnVat590.stCoeInterface.fRampTime_SP);
	fbCoeWrite.cbBufLen := SIZEOF(stVcnVat590.stCoeInterface.fRampTime_SP);
	fbCoeWrite.bExecute := TRUE;
ELSIF stVcnVat590.stCoeInterface.nRampMode_SP <> stCoeParameters.nRampMode_SP THEN
	fbCoeWrite.nIndex := cRampMode_SP.nIndex;
	fbCoeWrite.nSubIndex := cRampMode_SP.nSubIndex;
	fbCoeWrite.pSrcBuf := ADR(stVcnVat590.stCoeInterface.nRampMode_SP);
	fbCoeWrite.cbBufLen := SIZEOF(stVcnVat590.stCoeInterface.nRampMode_SP);
	fbCoeWrite.bExecute := TRUE;
ELSIF stVcnVat590.stCoeInterface.fPGain_SP <> stCoeParameters.fPGain_SP THEN
	fbCoeWrite.nIndex := cPGain_SP.nIndex;
	fbCoeWrite.nSubIndex := cPGain_SP.nSubIndex;
	fbCoeWrite.pSrcBuf := ADR(stVcnVat590.stCoeInterface.fPGain_SP);
	fbCoeWrite.cbBufLen := SIZEOF(stVcnVat590.stCoeInterface.fPGain_SP);
	fbCoeWrite.bExecute := TRUE;
END_IF

ftCoeWriteBusy(CLK:=fbCoeWrite.bBusy);
IF ftCoeWriteBusy.Q THEN
	fbCoeWrite.bExecute := FALSE;
	IF fbCoeWrite.bError THEN
		stVcnVat590.bCoeError := TRUE;
	END_IF
END_IF

fbCoeWrite();
END_ACTION

ACTION WriteToOutput:
(*Write to EPICS*)
stVcnVat590.bIlkOK := bExtIlkOK;
stVcnVat590.nPositionSP := REAL_TO_DINT(fCalcPosSP);
stVcnVat590.nPressureSP := REAL_TO_DINT(fCalcPresSP);
stVcnVat590.fReqPosition := fReqPos;
stVcnVat590.fReqPressure := fReqPres;
stVcnVat590.fPresSetLimit := fPresMaxLim;
stVcnVat590.fPosSetLimit := fUpperLimit;

(*Write to VAT valve*)
o_eCtrlModeSP := eValveModeSP;
o_nRawPositionSP := REAL_TO_DINT(fCalcPosSP);
o_nRawPressureSP := REAL_TO_DINT(fCalcPresSP);
o_stGenCtrlSP.Bit0ExecuteZero := stVcnVat590.bZero;
o_stGenCtrlSP.Bit4AccessMode := bRemAcsToggle;
END_ACTION

END_FUNCTION_BLOCK

// ---- POUs/Gauges/FB_IE514.TcPOU
(*This function is for the IE514 connected to controller IM540*)
(*This function provides ILK and Set Point Protection for the IE514*)
FUNCTION_BLOCK FB_IE514 EXTENDS FB_GaugeBase
VAR_IN_OUT
END_VAR
VAR_INPUT
	PG : ST_VG;
END_VAR
VAR_OUTPUT
	{attribute 'pytmc' := '
		pv:01
	'}
	IG_CH1 : ST_VG;
	{attribute 'pytmc' := '
		pv:02
	'}
	IG_CH2 : ST_VG; 
END_VAR
VAR
	rV : REAL; //Raw value in volts calculated from iTermBits
	rPRESS : REAL; //Calculated pressure from raw voltage
	tHvDis_CH1 : TON := (PT := T#20S); //HV turn on timer
	tHvDis_CH2 : TON := (PT := T#20S); //HV turn on timer
	
	rtHvSw_CH1 : R_TRIG;
	rtHvSw_CH2 : R_TRIG;
	
	tAction_CH1 : R_TRIG;
	tAction_CH2 : R_TRIG;	
	
	bCh1Sel : BOOL;
	bCh2Sel : BOOL;
	
	ePrevStateIG_CH1 : E_PressureState;
	ePrevStateIG_CH2 : E_PressureState;
	
	//rDefaultVAC_SP: REAL := 9E-3; // as per manual
	
	iTermBits : UINT := 30518; // The terminal's maximum value in bits default el3174 as per vacuum architecture
	binit : BOOL := TRUE;  // Do something at startup
	
	(*IOs to be linked*)
	/// Controls and I/Os
	i_iPRESS_R AT %I* : INT; // input raw pressure in bits (ADC) // 'TcLinkTo' (EL3174) ^Input
	q_xHV_DIS_CH1 AT %Q* : BOOL; // Enable Gauge High Voltage on CH1 when True // 'TcLinkTo' (EL2124) ^Output
	q_xHV_DIS_CH2 AT %Q* : BOOL; // Enable Gauge High Voltage on CH2 when True // 'TcLinkTo' (EL2124) ^Output
	i_xHV_ON AT %I*	: BOOL; // True when EMI is on  // 'TcLinkTo' (EL1004 or EL1008) ^Input
	i_xERR_CH1 AT %I* : BOOL; // TRUE when NO error is present on assigned channel
	i_xERR_CH2 AT %I* : BOOL; // TRUE when NO error is present on assigned channel
	i_xCH2_SEL AT %I* : BOOL; // TRUE when CH2 selected, FALSE when CH1 selected
END_VAR
VAR CONSTANT
	cMaxPressure : REAL := 7.5E-5; //Torr
	cMinPressure : REAL := 7.5E-14; //Torr
	cGaugeMinVoltage : REAL := 1.111; //minimum voltage corresponds to 7.5E-13 (7.498E-13)Torr which should be the minimum pressure IE514 can read.
	cGaugeMaxVoltage : REAL := 10.0; //maximum voltage corresponds 7.5E-5 Torr which should be the maximum pressure IE514 can read.
	cGaugeDisconnected : REAL := 10.2; //voltage when gauge is disconnected.
	cGaugeOff : REAL := 10.2; //voltage when gauge is turned off
	cDeadband : REAL := 0.05; //deadband in voltage
END_VAR
VAR PERSISTENT
    //Persistent variables for CH1
    rVAC_SP_CH1 : REAL;
	rPRO_SP_CH1 : REAL;
	rHYS_PR_CH1 : REAL;
    //Persistent variables for CH2
    rVAC_SP_CH2 : REAL;
	rPRO_SP_CH2 : REAL;
	rHYS_PR_CH2 : REAL;
END_VAR

(* 2-6-2023, Janez Govednik *)
(* This function will read the pressure from an IE514 gauge on an IM540. *)

(*Soft IO Linking*)
IO();

(*Select channel at the startup, according to input from the controller*)
IF bInit THEN
	IF NOT i_xCH2_SEL THEN
		bCh1Sel := TRUE;
		bCh2Sel := FALSE;
	ELSE
		bCh1Sel := FALSE;
		bCh2Sel := TRUE;
	END_IF
	bInit := FALSE;
END_IF

(*Only ONE channel can be turned ON at the same time*)
rtHvSw_CH1(CLK := IG_CH1.xHV_SW);
rtHvSw_CH2(CLK := IG_CH2.xHV_SW);
IF rtHvSw_CH1.Q THEN
	IG_CH2.xHV_SW := FALSE;
	IG_CH2.q_xHV_DIS := FALSE;
	bCh1Sel := TRUE;
	bCh2Sel := FALSE;
END_IF

IF rtHvSw_CH2.Q THEN
	IG_CH1.xHV_SW := FALSE;
	IG_CH1.q_xHV_DIS := FALSE;
	bCh1Sel := FALSE;
	bCh2Sel := TRUE;
END_IF

//Start timers when HV ON signal triggered
tHvDis_CH1(IN := IG_CH1.q_xHV_DIS, Q => IG_CH1.xTurnOnTime);
tHvDis_CH2(IN := IG_CH2.q_xHV_DIS, Q => IG_CH2.xTurnOnTime);

(*Raw voltage conversion*)
//check no div by zero
IF (iTermBits = 0) THEN iTermBits := 30518; END_IF
rV := 10*INT_TO_REAL(i_iPRESS_R)/iTermBits;

(*RAW voltage to Pressure conversion*)
rPRESS := LREAL_TO_REAL(EXPT(10, rV/10*LOG(cMaxPressure/cMinPressure) + LOG(cMinPressure))); //manual page 70 IM540 (Mode Full), (Scale) = Log
IF NOT i_xCH2_SEL THEN
	IG_CH1.rPRESS := rPRESS;
	IG_CH2.rPRESS := 0;
ELSE
	IG_CH2.rPRESS := rPRESS;
	IG_CH1.rPRESS := 0;
END_IF

(*Pressure gauge State checks*)
//CH1
IF bCh1Sel AND IG_CH1.xHV_SW THEN
	IF NOT i_xERR_CH1 THEN
		IG_CH1.eState := GaugeDisconnected;
		IG_CH1.rPRESS := 0;
	ELSIF rV <= cGaugeMaxVoltage AND rV >= cGaugeMinVoltage AND IG_CH1.i_xHV_ON THEN
		IG_CH1.eState := Valid; // NORMAL
	ELSIF rV >= 0.0 AND rV < cGaugeMinVoltage AND IG_CH1.i_xHV_ON THEN
		IG_CH1.eState := OoR; //Out of range according to manual
	ELSIF rV > cGaugeMaxVoltage AND rV < (cGaugeMaxVoltage + cDeadband) AND IG_CH1.i_xHV_ON THEN
		IG_CH1.eState := OoR; //Out of range according to manual
	ELSIF rV > (cGaugeMaxVoltage + cDeadband) AND tHvDis_CH1.Q THEN
		IG_CH1.eState := GaugeDisconnected; //gauge disconnected
		IG_CH1.rPRESS := 0;
	ELSIF rV > (cGaugeMaxVoltage + cDeadband) AND NOT tHvDis_CH1.Q THEN
		IG_CH1.eState := Starting; //gauge is starting
		IG_CH1.rPRESS := 0;
	ELSE
		IG_CH1.eState := PressInvalid; //other fault - could be no gauge, controller powering up etc.
		IG_CH1.rPRESS := 0;
	END_IF
ELSE
	IG_CH1.eState := Off; // Gauge turned OFF
	IG_CH1.rPRESS := 0;
END_IF

//CH2
IF bCh2Sel AND IG_CH2.xHV_SW THEN
	IF NOT i_xERR_CH2 THEN
		IG_CH2.eState := GaugeDisconnected;
		IG_CH2.rPRESS := 0;
	ELSIF rV <= cGaugeMaxVoltage AND rV >= cGaugeMinVoltage AND IG_CH2.i_xHV_ON THEN
		IG_CH2.eState := Valid; // NORMAL
	ELSIF rV >= 0.0 AND rV < cGaugeMinVoltage AND IG_CH2.i_xHV_ON THEN
		IG_CH2.eState := OoR; //Out of range according to manual
	ELSIF rV > cGaugeMaxVoltage AND rV < (cGaugeMaxVoltage + cDeadband) AND IG_CH2.i_xHV_ON THEN
		IG_CH2.eState := OoR; //Out of range according to manual
	ELSIF rV > (cGaugeMaxVoltage + cDeadband) AND tHvDis_CH2.Q THEN
		IG_CH2.eState := GaugeDisconnected; //gauge disconnected
		IG_CH2.rPRESS := 0;
	ELSIF rV > (cGaugeMaxVoltage + cDeadband) AND NOT tHvDis_CH2.Q THEN
		IG_CH2.eState := Starting; //gauge is starting
		IG_CH2.rPRESS := 0;
	ELSE
		IG_CH2.eState := PressInvalid; //other fault - could be no gauge, controller powering up etc.
		IG_CH2.rPRESS := 0;
	END_IF
ELSE
	IG_CH2.eState := Off; // Gauge turned OFF
	IG_CH2.rPRESS := 0;
END_IF

(* Ion Gauge Protection Functions *)
(* If the PG pressure is greater than the VG.PRO_SP then the gauge is disabled *)
(* If the PG pressure is less than the VG.PRO_SP then the gauge is enabled *)
(* This FB also implements some hysteresis so the gauge doesn't have rapid power cycling while near the turn on boundary *)

//CH1
IF (PG.rPRESS <= IG_CH1.rPRO_SP) THEN
	IG_CH1.q_xHV_DIS := IG_CH1.xHV_SW;
	IG_CH1.xILKOk := TRUE;
ELSIF IG_CH1.q_xHV_DIS AND tHvDis_CH1.Q THEN
	IF IG_CH1.rPRESS > (IG_CH1.rPRO_SP + IG_CH1.rHYS_PR) OR PG.rPRESS > (IG_CH1.rPRO_SP + IG_CH1.rHYS_PR) THEN
		IG_CH1.q_xHV_DIS := FALSE;
		IG_CH1.xHV_SW := FALSE;
	END_IF
ELSE 
	IG_CH1.q_xHV_DIS := FALSE;
	IG_CH1.xHV_SW := FALSE;
	IG_CH1.xILKOk := FALSE;
END_IF

//CH2
IF (PG.rPRESS <= IG_CH2.rPRO_SP) THEN
	IG_CH2.q_xHV_DIS := IG_CH2.xHV_SW;
	IG_CH2.xILKOk := TRUE;
ELSIF IG_CH2.q_xHV_DIS AND tHvDis_CH2.Q THEN
	IF IG_CH2.rPRESS > (IG_CH2.rPRO_SP + IG_CH2.rHYS_PR) OR PG.rPRESS > (IG_CH2.rPRO_SP + IG_CH2.rHYS_PR) THEN
		IG_CH2.q_xHV_DIS := FALSE;
		IG_CH2.xHV_SW := FALSE;
	END_IF
ELSE
	IG_CH2.q_xHV_DIS := FALSE;
	IG_CH2.xHV_SW := FALSE;
	IG_CH2.xILKOk := FALSE;
END_IF


(*Pressure gauge OK checks, Backwards compatibility*)
IG_CH1.xPRESS_OK := ((IG_CH1.eState = Valid) OR IG_CH1.xBAKEOUT);
IG_CH2.xPRESS_OK := ((IG_CH2.eState = Valid) OR IG_CH2.xBAKEOUT);

(*Setpoint evaluation*)
IG_CH1.xAT_VAC := IG_CH1.xPRESS_OK AND IG_CH1.rPRESS < IG_CH1.rVAC_SP;
IG_CH2.xAT_VAC := IG_CH2.xPRESS_OK AND IG_CH2.rPRESS < IG_CH2.rVAC_SP;

(*Logger*)
ACT_Logger();

(*Soft IO Linking*)
IO();

(*Load or save the persistent variables*)
ACT_Persistent();

ACTION ACT_Logger:
// ILK logger
(*CH1 of IM540 Controller*)
IF (IG_CH1.xLog) THEN
	IF NOT IG_CH1.xILKOk AND IG_CH1.q_xHV_DIS THEN
			fbLogger(sMsg:='Lost external interlock while gauge(CH1) was on.', eSevr:=TcEventSeverity.Critical);  	
	END_IF

	// Log Action
	tAction_CH1(CLK := IG_CH1.xHV_SW);
	IF tAction_CH1.Q THEN fbLogger(sMsg:='Ion gauge(CH1) commanded to switch on', eSevr:=TcEventSeverity.Info); END_IF

	//STATE Logger  
	IF ePrevStateIG_CH1 <> IG_CH1.eState THEN
		  CASE IG_CH1.eState OF
			ValidHi:
				fbLogger(sMsg:='Gauge(CH1) pressure valid high.', eSevr:=TcEventSeverity.Info);
			ValidLo:
				fbLogger(sMsg:='Gauge(CH1) pressure valid low.', eSevr:=TcEventSeverity.Info);
			Valid:
				fbLogger(sMsg:='Gauge(CH1) pressure valid.', eSevr:=TcEventSeverity.Info);
			GaugeDisconnected:
				fbLogger(sMsg:='Gauge(CH1) Disconnected.', eSevr:=TcEventSeverity.Critical);
			PressInvalid:
				fbLogger(sMsg:='Gauge(CH1) pressure invalid.', eSevr:=TcEventSeverity.Warning);
			OoR:
				fbLogger(sMsg:='Gauge(CH1) pressure out of range.', eSevr:=TcEventSeverity.Warning);
			Starting:
				fbLogger(sMsg:='Gauge(CH1) starting.', eSevr:=TcEventSeverity.Info);
		  END_CASE
		  ePrevStateIG_CH1 := IG_CH1.eState;
	  END_IF
END_IF
  
(*CH2 of IM540 Controller*)
IF (IG_CH2.xLog) THEN
	IF NOT IG_CH2.xILKOk AND IG_CH2.q_xHV_DIS THEN
			fbLogger(sMsg:='Lost external interlock while gauge(CH2) was on.', eSevr:=TcEventSeverity.Critical);  	
	END_IF

	// Log Action
	tAction_CH2(CLK := IG_CH2.xHV_SW);
	IF tAction_CH2.Q THEN fbLogger(sMsg:='Ion gauge(CH2) commanded to switch on', eSevr:=TcEventSeverity.Info); END_IF

	//STATE Logger  
	IF ePrevStateIG_CH2 <> IG_CH2.eState THEN
		  CASE IG_CH2.eState OF
			ValidHi:
				fbLogger(sMsg:='Gauge(CH2) pressure valid high.', eSevr:=TcEventSeverity.Info);
			ValidLo:
				fbLogger(sMsg:='Gauge(CH2) pressure valid low.', eSevr:=TcEventSeverity.Info);
			Valid:
				fbLogger(sMsg:='Gauge(CH2) pressure valid.', eSevr:=TcEventSeverity.Info);
			GaugeDisconnected:
				fbLogger(sMsg:='Gauge(CH2) Disconnected.', eSevr:=TcEventSeverity.Critical);
			PressInvalid:
				fbLogger(sMsg:='Gauge(CH2) pressure invalid.', eSevr:=TcEventSeverity.Warning);
			OoR:
				fbLogger(sMsg:='Gauge(CH2) pressure out of range.', eSevr:=TcEventSeverity.Warning);
			Starting:
				fbLogger(sMsg:='Gauge(CH2) starting.', eSevr:=TcEventSeverity.Info);
		  END_CASE
		  ePrevStateIG_CH2 := IG_CH2.eState;
	  END_IF
END_IF
END_ACTION

ACTION ACT_Persistent:
(*On first PLC pass, load the persistent value into the structrue variable*)
IF (SUPER^.bRestorePersistentData) THEN
	SUPER^.bRestorePersistentData := FALSE;
    //CH1
	IF (rVAC_SP_CH1 <> 0) THEN
		IG_CH1.rVAC_SP := rVAC_SP_CH1;
	END_IF;
	IF (rPRO_SP_CH1 <> 0) THEN
		IG_CH1.rPRO_SP := rPRO_SP_CH1;
	END_IF;
	IF (rHYS_PR_CH1 <> 0) THEN
		IG_CH1.rHYS_PR := rHYS_PR_CH1;
	END_IF;
    //CH2
	IF (rVAC_SP_CH2 <> 0) THEN
		IG_CH2.rVAC_SP := rVAC_SP_CH2;
	END_IF;
	IF (rPRO_SP_CH2 <> 0) THEN
		IG_CH2.rPRO_SP := rPRO_SP_CH2;
	END_IF;
	IF (rHYS_PR_CH2 <> 0) THEN
		IG_CH2.rHYS_PR := rHYS_PR_CH2;
	END_IF;
END_IF
(*Check if a new value has been written in the structure variable copy it to the persistent variable*)
//CH1
IF NOT (IG_CH1.rVAC_SP = rVAC_SP_CH1)  THEN
	rVAC_SP_CH1 := IG_CH1.rVAC_SP;
END_IF;

IF NOT (IG_CH1.rPRO_SP = rPRO_SP_CH1) THEN
	rPRO_SP_CH1 := IG_CH1.rPRO_SP;
END_IF;

IF NOT (IG_CH1.rHYS_PR = rHYS_PR_CH1) THEN
	rHYS_PR_CH1 := IG_CH1.rHYS_PR;
END_IF;

//CH2
IF NOT (IG_CH2.rVAC_SP = rVAC_SP_CH2)  THEN
	rVAC_SP_CH2 := IG_CH2.rVAC_SP;
END_IF;

IF NOT (IG_CH2.rPRO_SP = rPRO_SP_CH2) THEN
	rPRO_SP_CH2 := IG_CH2.rPRO_SP;
END_IF;

IF NOT (IG_CH2.rHYS_PR = rHYS_PR_CH2) THEN
	rHYS_PR_CH2 := IG_CH2.rHYS_PR;
END_IF;
END_ACTION

ACTION IO:
(*soft link inputs*)
IF NOT i_xCH2_SEL THEN
	IG_CH1.i_iPRESS_R := i_iPRESS_R;
	IG_CH1.i_xHV_ON := i_xHV_ON;
	IG_CH2.i_iPRESS_R := 0;
	IG_CH2.i_xHV_ON := FALSE;
ELSE
	IG_CH2.i_iPRESS_R := i_iPRESS_R;
	IG_CH2.i_xHV_ON := i_xHV_ON;
	IG_CH1.i_iPRESS_R := 0;
	IG_CH1.i_xHV_ON := FALSE;
END_IF

(*soft link outputs*)
q_xHV_DIS_CH1 := IG_CH1.q_xHV_DIS;
q_xHV_DIS_CH2 := IG_CH2.q_xHV_DIS;

IG_CH1.sPath := sPath;
IG_CH2.sPath := sPath;
END_ACTION

METHOD M_AutoOnCh1 : BOOL
VAR_INPUT
END_VAR
this^.IG_CH1.q_xHV_DIS := TRUE;
END_METHOD

METHOD M_AutoOnCh2 : BOOL
VAR_INPUT
END_VAR
this^.IG_CH2.q_xHV_DIS := TRUE;
END_METHOD

METHOD M_HVECh1 : BOOL
VAR_INPUT
		enable : BOOL; // set to true to enable, false to disable;
END_VAR
this^.IG_CH1.xHV_SW := (enable);
END_METHOD

METHOD M_HVECh2 : BOOL
VAR_INPUT
		enable : BOOL; // set to true to enable, false to disable;
END_VAR
this^.IG_CH2.xHV_SW := (enable);
END_METHOD

METHOD M_SetBits
VAR_INPUT
	TermBits : UINT; // The beckhoff terminal's maximum value in bits
END_VAR
this^.iTermBits := TermBits;
END_METHOD

END_FUNCTION_BLOCK

// ---- POUs/Gauges/FB_MX7M.TcPOU
(* This function is for the Cold Cathode MX7M from Televac. *)
(*This function provides ILK and Set Point Protection for the Cold Cathode*)
FUNCTION_BLOCK FB_MX7M EXTENDS FB_GaugeBase
VAR_IN_OUT
		
END_VAR
VAR_INPUT
	PG : ST_VG;
	tRecoverDelay : TIME := T#600S; (*Delay Time after the first cycle to start the device. Default is 600S*)
END_VAR
VAR_OUTPUT
    {attribute 'pytmc' := '
    pv: 
	'}
	IG : ST_VG;
END_VAR
VAR
	rV : REAL; //Calculated raw voltage from ADC on analog input
	rPress : REAL; //Calculated pressure
	tGaugeTurnOnTmr : TON;
	iTermBits : UINT := 30518 ; //The terminal's maximum value in bits
	bInit : BOOL := TRUE;
	rVIntPart : INT;
	rVFracPart : REAL;
	(*IOs to be linked*)
	//Controls and I/Os
	i_iPRESS_R AT %I* : INT; //Pressure reading // 'TcLinkTo' (EL3174-0002 or EP3174-0002)^Input
	q_xHV_DIS AT %Q* : BOOL; //Enable High Voltage when True // 'TcLinkTo' (EL2624 or EP2624-0002)^Output
END_VAR
VAR CONSTANT
	//Ranges ~1.5 to ~10.1 Vdc (5E-11 to 1E-2)
	//Must set the analog output scaling to Linear by Decade!!
	cGaugeMinV : REAL := 1.5;
	cGaugeMaxV : REAL := 10.1;
	cGaugeStartingV : REAL := 10.5;
	cDefaultPressure : REAL := 0.0;
	cDeadband : REAL := 0.1;
END_VAR
VAR PERSISTENT
	bWasOn : BOOL;
	bAutoRecover : BOOL;
	bAutoRecoverWrite : BOOL;
END_VAR

(*Calculate raw voltage*)
IF (iTermBits = 0) THEN iTermBits := 30518; END_IF
rV := 10*INT_TO_REAL(i_iPRESS_R)/iTermBits;

(*Calculate pressure*)
rVIntPart := TRUNC_INT(rV); // Get the integer part
rVFracPart := rV - INT_TO_REAL(rVIntPart); // Get the fractional part
rPRESS := rVFracPart*LREAL_TO_REAL(EXPT(10,(rVIntPart-11)));

(*Set Guage State based on the Analog voltage*)
IF IG.q_xHV_DIS THEN
    IF rV >= cGaugeMinV AND rV <= cGaugeMaxV THEN
		IG.eState := Valid;
	    IG.rPRESS := rPRESS;
    ELSIF rV > cGaugeStartingV - cDeadband THEN
	    IG.eState := Starting;
	    IG.rPRESS := cDefaultPressure;
    ELSIF rV < cGaugeMinV - cDeadband THEN
	    IG.eState := GaugeDisconnected;
	    IG.rPRESS := cDefaultPressure;
    ELSIF rV > cGaugeMaxV AND rV < cGaugeStartingV - cDeadband THEN
	    IG.eState := OoR;
	    IG.rPRESS := cDefaultPressure;
	ELSE
	    IG.eState := PressInvalid;
	    IG.rPRESS := cDefaultPressure;
    END_IF
ELSE
	IG.eState := Off;
	IG.rPRESS := cDefaultPressure;
END_IF


(*
IF rV <= vDisconnected AND IG.q_xHV_DIS THEN
	IG.eState := ValidLo;
	IG.rPRESS := rMinPressure;
ELSIF rV <= vDisconnected AND NOT IG.q_xHV_DIS THEN
	IG.eState := GaugeDisconnected;
	IG.rPRESS := cDefaultPressure;
ELSIF rV > vDisconnected AND rV <= vGaugeMax AND IG.q_xHV_DIS THEN
	IG.eState := Valid;
	IG.rPRESS := rPRESS;
ELSIF rV > vGaugeMax AND rV < (vGaugeOff - rDeadband) AND IG.q_xHV_DIS THEN
	IG.eState := OoR;
	IG.rPRESS := cDefaultPressure;
ELSIF rV > (vGaugeOff - rDeadband) AND IG.q_xHV_DIS THEN
	IG.eState := Starting;
	IG.rPRESS := cDefaultPressure;
ELSIF rV > vGaugeOff - rDeadband AND NOT IG.q_xHV_DIS THEN
	IG.eState := Off;
	IG.rPRESS := cDefaultPressure;
ELSE
	IG.eState := PressInvalid;
	IG.rPRESS := cDefaultPressure;
END_IF
*)

(* Ion Gauge Protection Functions *)
(* If the PG pressure is greater than the VG.PRO_SP then the gauge is disabled *)
(* If the PG pressure is less than the VG.PRO_SP then the gauge is enabled *)
(* This FB also implements some hysteresis so the gauge doesn't have rapid power cycling while near the turn on boundary *)
IF PG.rPRESS <= IG.rPRO_SP AND PG.xPRESS_OK THEN
	IG.q_xHV_DIS := IG.xHV_SW;
	IG.xILKOk := TRUE;
ELSIF IG.q_xHV_DIS THEN
	IF IG.rPRESS > (IG.rPRO_SP + IG.rHYS_PR)  OR PG.rPRESS > (IG.rPRO_SP + IG.rHYS_PR) THEN
		IG.q_xHV_DIS := FALSE;
		IG.xHV_SW := FALSE;
	END_IF
ELSE
	IG.q_xHV_DIS := FALSE;
	IG.xHV_SW := FALSE;
	IG.xILKOk := FALSE;
END_IF


(*Pressure gauge OK checks*)
tGaugeTurnOnTmr(IN:=IG.q_xHV_DIS, PT:=T#10S, Q=>IG.xTurnOnTime);

//Backwards compatibility
IG.xPRESS_OK := (IG.eState = Valid) OR IG.xBAKEOUT;

(*Setpoint evaluation*)
IG.xAT_VAC := (IG.xPRESS_OK AND (IG.rPRESS < IG.rVAC_SP)) OR IG.xBAKEOUT AND (IG.eState = Valid);

(*Logging*)
ACT_Logger();

(*Soft IO Linking*)
IO();

(*Load or save the persistent variables*)
ACT_Persistent();

(*Run Auto Recovery*)
ACT_Recover();

ACTION ACT_Logger:
// ILK logger
IF (IG.xLog) THEN
	IF NOT IG.xILKOk AND IG.q_xHV_DIS THEN
			fbLogger(sMsg:='Lost external interlock while gauge was on.', eSevr:=TcEventSeverity.Critical);  	
	END_IF
	
	
	// Log Action
	tAction(CLK := IG.xHV_SW);
	IF tAction.Q THEN fbLogger(sMsg:='Ion gauge commanded to switch on', eSevr:=TcEventSeverity.Info); END_IF
	
	
	
	//STATE Logger  
	IF ePrevState <> IG.eState THEN
		  CASE IG.eState OF
			ValidHi:
				fbLogger(sMsg:='Gauge pressure valid high.', eSevr:=TcEventSeverity.Info);
			ValidLo:
				fbLogger(sMsg:='Gauge pressure valid low.', eSevr:=TcEventSeverity.Info);
			Valid:
				fbLogger(sMsg:='Gauge pressure valid.', eSevr:=TcEventSeverity.Info);
			GaugeDisconnected:
				fbLogger(sMsg:='Gauge Disconnected.', eSevr:=TcEventSeverity.Critical);
			PressInvalid:
				fbLogger(sMsg:='Gauge pressure invalid.', eSevr:=TcEventSeverity.Warning);
			OoR:
				fbLogger(sMsg:='Gauge pressure out of range.', eSevr:=TcEventSeverity.Warning);
			Starting:
				fbLogger(sMsg:='Gauge starting.', eSevr:=TcEventSeverity.Info);
		  END_CASE
      ePrevState := IG.eState;  
	  END_IF
END_IF
END_ACTION

ACTION ACT_Persistent:
(*On first PLC pass, load the persistent value into the structrue variable*)
IF (SUPER^.bRestorePersistentData) THEN
	SUPER^.bRestorePersistentData := FALSE;
	IF (rVAC_SP <> 0) THEN
		IG.rVAC_SP := rVAC_SP;
	END_IF;
	IF (rPRO_SP <> 0) THEN
		IG.rPRO_SP := rPRO_SP;
	END_IF;
	IF (rHYS_PR <> 0) THEN
		IG.rHYS_PR := rHYS_PR;
	END_IF;
	IF (bAutoRecoverWrite) THEN
		IG.xAutoOn := bAutoRecover;
	END_IF;
END_IF
(*Check if a new value has been written in the structure variable copy it to the persistent variable*)
IF NOT (IG.rVAC_SP = rVAC_SP)  THEN
	rVAC_SP := IG.rVAC_SP;
END_IF;

IF NOT (IG.rPRO_SP = rPRO_SP) THEN
	rPRO_SP := IG.rPRO_SP;
END_IF;

IF NOT (IG.rHYS_PR = rHYS_PR) THEN
	rHYS_PR := IG.rHYS_PR;
END_IF;

IF NOT(bAutoRecoverWrite) OR NOT (bAutoRecover = IG.xAutoOn) THEN
	bAutoRecover := IG.xAutoOn;
	bAutoRecoverWrite := TRUE;
END_IF;

stateTimer(PT := T#10S);
IF (stateTimer.Q) THEN
	bWasOn := (IG.eState >= Valid);
	stateTimer.IN := FALSE;
	fbWritePersistentData(NETID:='', PORT:=851, START:=TRUE, TMOUT:=T#1s);
END_IF;
END_ACTION

ACTION ACT_Recover:
fbGetCurTaskIdx();
IF (TwinCAT_SystemInfoVarList._TaskInfo[fbGetCurTaskIdx.index].FirstCycle) THEN
	tRecover.IN := TRUE;
END_IF
tRecover(PT := tRecoverDelay);
IF NOT(bAutoRecoverWrite) OR (tRecover.Q AND bAutoRecover) THEN
	This^.M_Recover();
	tRecover.IN := FALSE;
END_IF
END_ACTION

ACTION IO:
(*soft link inputs*)
IG.i_iPRESS_R := i_iPRESS_R; 
IG.i_xHV_ON := IG.q_xHV_DIS;  //not a real readback, assuming turning on HV output, HV status is ON and vice versa

(*soft link outputs*)
q_xHV_DIS := IG.q_xHV_DIS;

(*Gauge name link*)
IG.sPath := sPath;
END_ACTION

METHOD M_HVE : BOOL
VAR_INPUT
		bEnable : BOOL; // set to true to enable, false to disable;
END_VAR
this^.IG.xHV_SW := bEnable;
END_METHOD

METHOD M_Recover : BOOL
VAR_INPUT
END_VAR
This^.M_HVE(This^.bWasOn);
M_Recover := bWasOn;
IF (bWasOn) THEN fbLogger(sMsg:='Auto Recovery Initiated.', eSevr:=TcEventSeverity.Info); END_IF;
END_METHOD

METHOD M_SetBits : BOOL
VAR_INPUT
	TermBits : UINT; // The terminal's maximum value in bits
END_VAR
This^.iTermBits := TermBits;
END_METHOD

END_FUNCTION_BLOCK

// ---- POUs/CoE/FB_CoE_Read.TcPOU
FUNCTION_BLOCK FB_CoE_Read
VAR_INPUT
	// Link this to your terminal's drive reference variables under InfoData.
	stPlcDriveRef : ST_PlcDriveRef;
END_VAR
VAR_OUTPUT
END_VAR
VAR
	// Read Error
	bReadError : BOOL;
	// Data successfully received
	bDataReceived : BOOL := FALSE;
	
	fbCoeRead: FB_CoERead_ByDriveRef;
	
	stDriveRef: ST_DriveRef;
	
	nState : BYTE := 0;   //State Machine
END_VAR

stDriveRef.sNetId := F_CreateAmsNetId(stPlcDriveRef.aNetId);
stDriveRef.nSlaveAddr := stPlcDriveRef.nSlaveAddr;
stDriveRef.nDriveNo := stPlcDriveRef.nDriveNo;
stDriveRef.nDriveType := stPlcDriveRef.nDriveType;

CASE nState OF
	0: //Idle state
		HandleIdle();
	10: //Reading data
		HandleReadingData();
	100: //Handle Error
		HandleError();
END_CASE

ACTION HandleError:
// wait for reset ccmmand
bDataReceived := FALSE;
END_ACTION

ACTION HandleIdle:
fbCoeRead(bExecute := FALSE);
// Reset Data received bit
bDataReceived := FALSE;
END_ACTION

ACTION HandleReadingData:
fbCoeRead(bExecute := TRUE);        // Execute CoE read until done
IF fbCoeRead.bError THEN
	nState := 100;     // Error case
	bReadError := TRUE;
ELSE
	IF NOT fbCoeRead.bBusy THEN
         nState := 0;    // Done
		 bDataReceived := TRUE;
	END_IF
END_IF
END_ACTION

METHOD InErrorState : BOOL
VAR_INPUT
END_VAR
IF nState = 100 THEN
	InErrorState := TRUE;
ELSE
	InErrorState := FALSE;
END_IF
END_METHOD

METHOD IsBusy : BOOL
VAR_INPUT
END_VAR
IF nState <> 0 THEN
	IsBusy := TRUE;
ELSE
	IsBusy := FALSE;
END_IF
END_METHOD

PROPERTY IsDataReceived : BOOL
GET
IsDataReceived := bDataReceived;
END_GET
END_PROPERTY

METHOD ReadData
VAR_INPUT
	//stCoeParameter : ST_CoeParameter;
	nIndex: WORD;
	// Hexadecimal subindex of CoE, e.g. the 12 in 8010:12
	nSubIndex: BYTE;
	// Pointer to a value to fill with the result of the read, e.g. ADR(MyValue)
	pDstBuf: PVOID;
	// Data size of pDstBuf, e.g. SIZEOF(MyValue)
	cbBufLen: UDINT;
END_VAR
IF nState <> 0 THEN
	RETURN;
END_IF

fbCoeRead(
	stDriveRef := stDriveRef,
	nIndex := nIndex,
	nSubIndex := nSubIndex,
	pDstBuf := pDstBuf,
	cbBufLen := cbBufLen,
	tTimeout := T#1S,
);

// Go to Reading data state
nState := 10;
END_METHOD

METHOD ResetError
VAR_INPUT
END_VAR
IF nState <> 100 THEN
	RETURN;
END_IF

// Reset read error
bReadError := FALSE;
// Go to Idle state
nState := 0;
END_METHOD

END_FUNCTION_BLOCK

// ---- POUs/CoE/FB_CoE_Write.TcPOU
FUNCTION_BLOCK FB_CoE_Write
VAR_INPUT
	// Link this to your terminal's drive reference variables under InfoData.
	stPlcDriveRef : ST_PlcDriveRef;
END_VAR
VAR_OUTPUT
END_VAR
VAR
	// Write Error
	bWriteError : BOOL;
	// Data successfully sent
	bDataSent : BOOL := FALSE;
	
	fbCoeWrite: FB_CoEWrite_ByDriveRef;
	
	stDriveRef: ST_DriveRef;
	
	nState : BYTE := 0;   //State Machine
END_VAR

stDriveRef.sNetId := F_CreateAmsNetId(stPlcDriveRef.aNetId);
stDriveRef.nSlaveAddr := stPlcDriveRef.nSlaveAddr;
stDriveRef.nDriveNo := stPlcDriveRef.nDriveNo;
stDriveRef.nDriveType := stPlcDriveRef.nDriveType;

CASE nState OF
	0: //Idle state
		HandleIdle();
	1: //Writing data
		HandleWritingData();
	100: //Handle Error
		HandleError();
END_CASE

ACTION HandleError:
// wait for reset ccmmand
bDataSent := FALSE;
END_ACTION

ACTION HandleIdle:
fbCoeWrite(bExecute := FALSE);
// Reset DataSent bit
bDataSent := FALSE;
END_ACTION

ACTION HandleWritingData:
fbCoeWrite(bExecute := TRUE);       // Execute CoE write until done
IF fbCoeWrite.bError THEN
	nState := 100;     // Error case
	bWriteError := TRUE;
ELSE
	IF NOT fbCoeWrite.bBusy THEN
		nState := 0;    // Done
		bDataSent := TRUE;
	END_IF
END_IF
END_ACTION

METHOD InErrorState : BOOL
VAR_INPUT
END_VAR
IF nState = 100 THEN
	InErrorState := TRUE;
ELSE
	InErrorState := FALSE;
END_IF
END_METHOD

METHOD IsBusy : BOOL
VAR_INPUT
END_VAR
IF nState <> 0 THEN
	IsBusy := TRUE;
ELSE
	IsBusy := FALSE;
END_IF
END_METHOD

PROPERTY IsDataSent : BOOL
GET
IsDataSent := bDataSent;
END_GET
END_PROPERTY

METHOD ResetError
VAR_INPUT
END_VAR
IF nState <> 100 THEN
	RETURN;
END_IF

// Reset write error
bWriteError := FALSE;
// Go to Idle state
nState := 0;
END_METHOD

METHOD WriteData
VAR_INPUT
	//stCoeParameter : ST_CoeParameter;
	nIndex: WORD;
	// Hexadecimal subindex of CoE, e.g. the 12 in 8010:12
	nSubIndex: BYTE;
	// Pointer to a value to fill with the result of the read, e.g. ADR(MyValue)
	pSrcBuf: PVOID;
	// Data size of pSrcBuf, e.g. SIZEOF(MyValue)
	cbBufLen: UDINT;
END_VAR
IF nState <> 0 THEN
	RETURN;
END_IF

fbCoeWrite(
	stDriveRef := stDriveRef,
	nIndex := nIndex,
	nSubIndex := nSubIndex,
	pSrcBuf := pSrcBuf,
	cbBufLen := cbBufLen,
	tTimeout := T#1S,
);

// Go to Writing Data state
nState := 1;
END_METHOD

END_FUNCTION_BLOCK
